PROGRAM com_task
VAR
END_VAR

(* Zähler *)
Zaehler();

END_PROGRAM

(* stored: Version 1.1.0.1, ProductVersion 3.1.4024.10
   POU com_task: Id {2a6820b0-4f66-4d85-a976-c6f73a5f0ae5}, SpecialFunc None *)
